(* Logix 5000 project; controller Machine_Maintenance_Lab2 vendor 1 type 14 code 155 rev 36.11; software revision 36.00 *)

TASK MainTask (continuous, watchdog 500 ms) : MainProgram

MODULES
   Local : vendor 1 type 14 code 155 (PointIO 0, rev 36.11)
      Discrete_IO : Embedded (PointIO 1, rev 36.11, Output RPI 20 ms)
END_MODULES

PROGRAM MainProgram   (* main routine MainRoutine *)
VAR
   counter : COUNTER := (PRE := 5);
   CycleCounter : COUNTER := (PRE := 5);
   delay : TIMER := (PRE := 10);
   HighCycleTimer : COUNTER := (PRE := 700);
   i_CycleDone : ALIAS FOR o_CycleDone;
   i_GreenPB : ALIAS FOR Local:1:I.Data.0;
   i_GreenPB_ConveyorStart : ALIAS FOR i_GreenPB;
   i_GreenPBLight_Conveyor1ON : ALIAS FOR o_GreenPBLight_Conveyor1ON;
   i_Pause : ALIAS FOR Pause;
   i_Piston : ALIAS FOR Local:1:O.Data.2;
   i_RedPB_StopButton : ALIAS FOR Local:1:I.Data.1;
   i_RedPBLight_Conveyor2ON : ALIAS FOR o_RedPBLight_Conveyor2ON;
   i_Turnkey : ALIAS FOR Local:1:I.Data.2;
   i_Turnkey_ItemSensor : ALIAS FOR i_Turnkey;
   ItemCounter1 : COUNTER := (PRE := 5);
   ItemCounterLeft : COUNTER := (PRE := 5);
   ItemCounterRight : COUNTER := (PRE := 6);
   LowCycleTimer : COUNTER := (PRE := 300);
   MotorDelay : TIMER := (PRE := 1000);
   MotorDelay1 : TIMER := (PRE := 1000);
   NewCycle : BOOL;
   o_CycleDone : BOOL;
   o_GreenPBLight : ALIAS FOR Local:1:O.Data.0;
   o_GreenPBLight_Conveyor1ON : ALIAS FOR o_GreenPBLight;
   o_motorOup3 : ALIAS FOR Local:1:O.Data.3;
   o_motorOup4 : ALIAS FOR Local:1:O.Data.4;
   o_Piston : ALIAS FOR i_Piston;
   o_RedPBLight : ALIAS FOR Local:1:O.Data.1;
   o_RedPBLight_Conveyor2ON : ALIAS FOR o_RedPBLight;
   OS_Out : BOOL;
   Pause : BOOL;
   ResetDelay : TIMER := (PRE := 500);
   Start : BOOL;
   ThreeSecTimer : TIMER := (PRE := 3000);
   timer : TIMER := (PRE := 5000);
   TimerHighCycle : TIMER := (PRE := 700);
   TimerLowCycle : TIMER := (PRE := 300);
   TurnkeyOneShot : BOOL;
   TurnkeyOneShot2 : BOOL;
END_VAR

ROUTINE MainRoutine   (* ladder *)
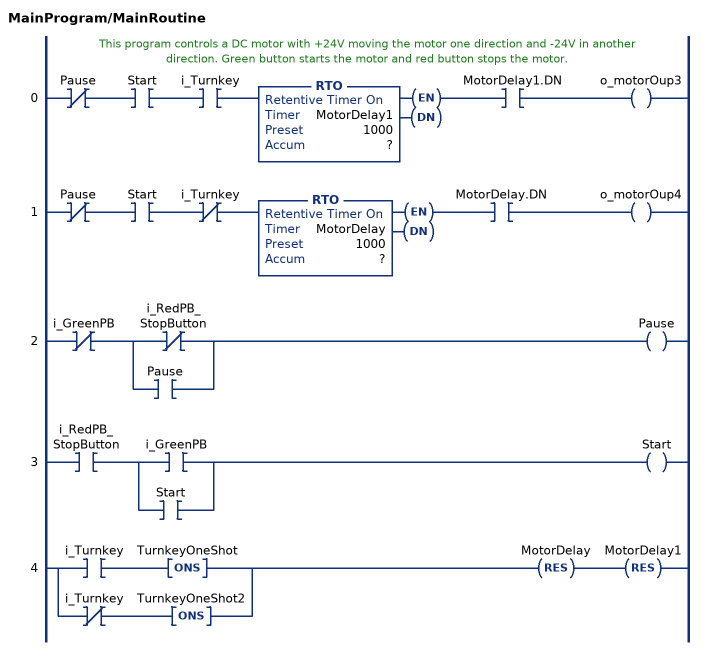
   // This program controls a DC motor with +24V moving the motor one direction and -24V in another direction. Green button starts the motor and red button stops the motor.
   0: XIO(Pause)XIC(Start)XIC(i_Turnkey)RTO(MotorDelay1,?,?)XIC(MotorDelay1.DN)OTE(o_motorOup3);
   1: XIO(Pause)XIC(Start)XIO(i_Turnkey)RTO(MotorDelay,?,?)XIC(MotorDelay.DN)OTE(o_motorOup4);
   2: XIO(i_GreenPB)[XIO(i_RedPB_StopButton) ,XIC(Pause) ]OTE(Pause);
   3: XIC(i_RedPB_StopButton)[XIC(i_GreenPB) ,XIC(Start) ]OTE(Start);
   4: [XIC(i_Turnkey) ONS(TurnkeyOneShot) ,XIO(i_Turnkey) ONS(TurnkeyOneShot2) ]RES(MotorDelay)RES(MotorDelay1);
END_ROUTINE
END_PROGRAM
